FUNCTION_BLOCK MainTank (* Basic Function Block Type *)
  (* Standard: 61499-2 *)
  (* Version 0.0, 2019-06-19, 4DIAC-IDE, 4DIAC-Consortium *)
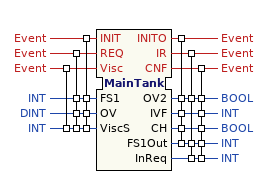
  EVENT_INPUT
    INIT WITH FS1, ViscS, OV; (* Initialization Request *)
    REQ WITH FS1, ViscS, OV; (* Normal Execution Request *)
    Visc WITH ViscS;
  END_EVENT
  EVENT_OUTPUT
    INITO WITH OV2, IVF, CH, FS1Out; (* Initialization Confirm *)
    IR WITH OV2, InReq, FS1Out; (* In flow request *)
    CNF WITH OV2, IVF, CH, InReq, FS1Out;
  END_EVENT
  VAR_INPUT
    FS1 : INT; (* Fluid Level Sensor *)
    OV : DINT; (* Temperature Sensor *)
    ViscS : INT; (* Viscosity Status *)
  END_VAR
  VAR_OUTPUT
    OV2 : BOOL; (* Outlet valve *)
    IVF : INT;
    CH : BOOL; (* Cartridge Heater *)
    FS1Out : INT;
    InReq : INT; (* Inlet Request *)
  END_VAR
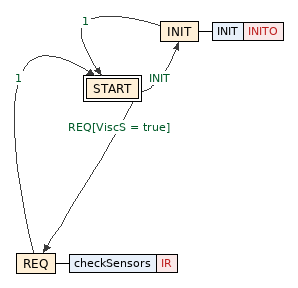
  EC_STATES
    START; (* Initial State *)
    INIT : INIT -> INITO; (* Initialization *)
    REQ : checkSensors -> IR; (* Normal execution *)
  END_STATES
  EC_TRANSITIONS
    START TO INIT := INIT;
    INIT TO START := 1;
    START TO REQ := REQ[ViscS = true];
    REQ TO START := 1;
  END_TRANSITIONS
  ALGORITHM INIT IN ST: (* Initialization algorithm *)

  END_ALGORITHM
  ALGORITHM checkSensors IN ST: (* new algorithm *)
IF ViscS = 1 THEN
	IF FS1 < 70 THEN
		InReq := 1;
	END_IF;
END_IF;
  END_ALGORITHM
END_FUNCTION_BLOCK
